(* IEC 61131-3 sources: UniTest/UniTest_br/Library_tests/main, 1 file *)

(* ---- main.st ---- *)
PROGRAM _CYCLIC
    (*https://github.com/tkucic/UniTest/blob/main/docs/docs/ns/Library_tests/prg/main.md*)
    testReporter(Results:=gResults);
END_PROGRAM
